(* PLC project Unnamed, Unknown Unnamed 1 *)
(* stored: creationDateTime 2025-06-21T03:07:53, modificationDateTime 2025-06-21T03:50:31 *)

PROGRAM ctud_pou
  VAR
    input1 AT %IX100.0 : BOOL;
    input2 AT %IX100.1 : BOOL;
    reset AT %IX100.2 : BOOL;
    load AT %IX100.3 : BOOL;
    output1 AT %QX100.0 : BOOL;
    output2 AT %QX100.1 : BOOL;
  END_VAR
  VAR
    CTUD0 : CTUD;
  END_VAR
  VAR  (* added by the conversion: wires and edge detectors of the diagram *)
    R_TRIG1 : R_TRIG;
    R_TRIG2 : R_TRIG;
  END_VAR

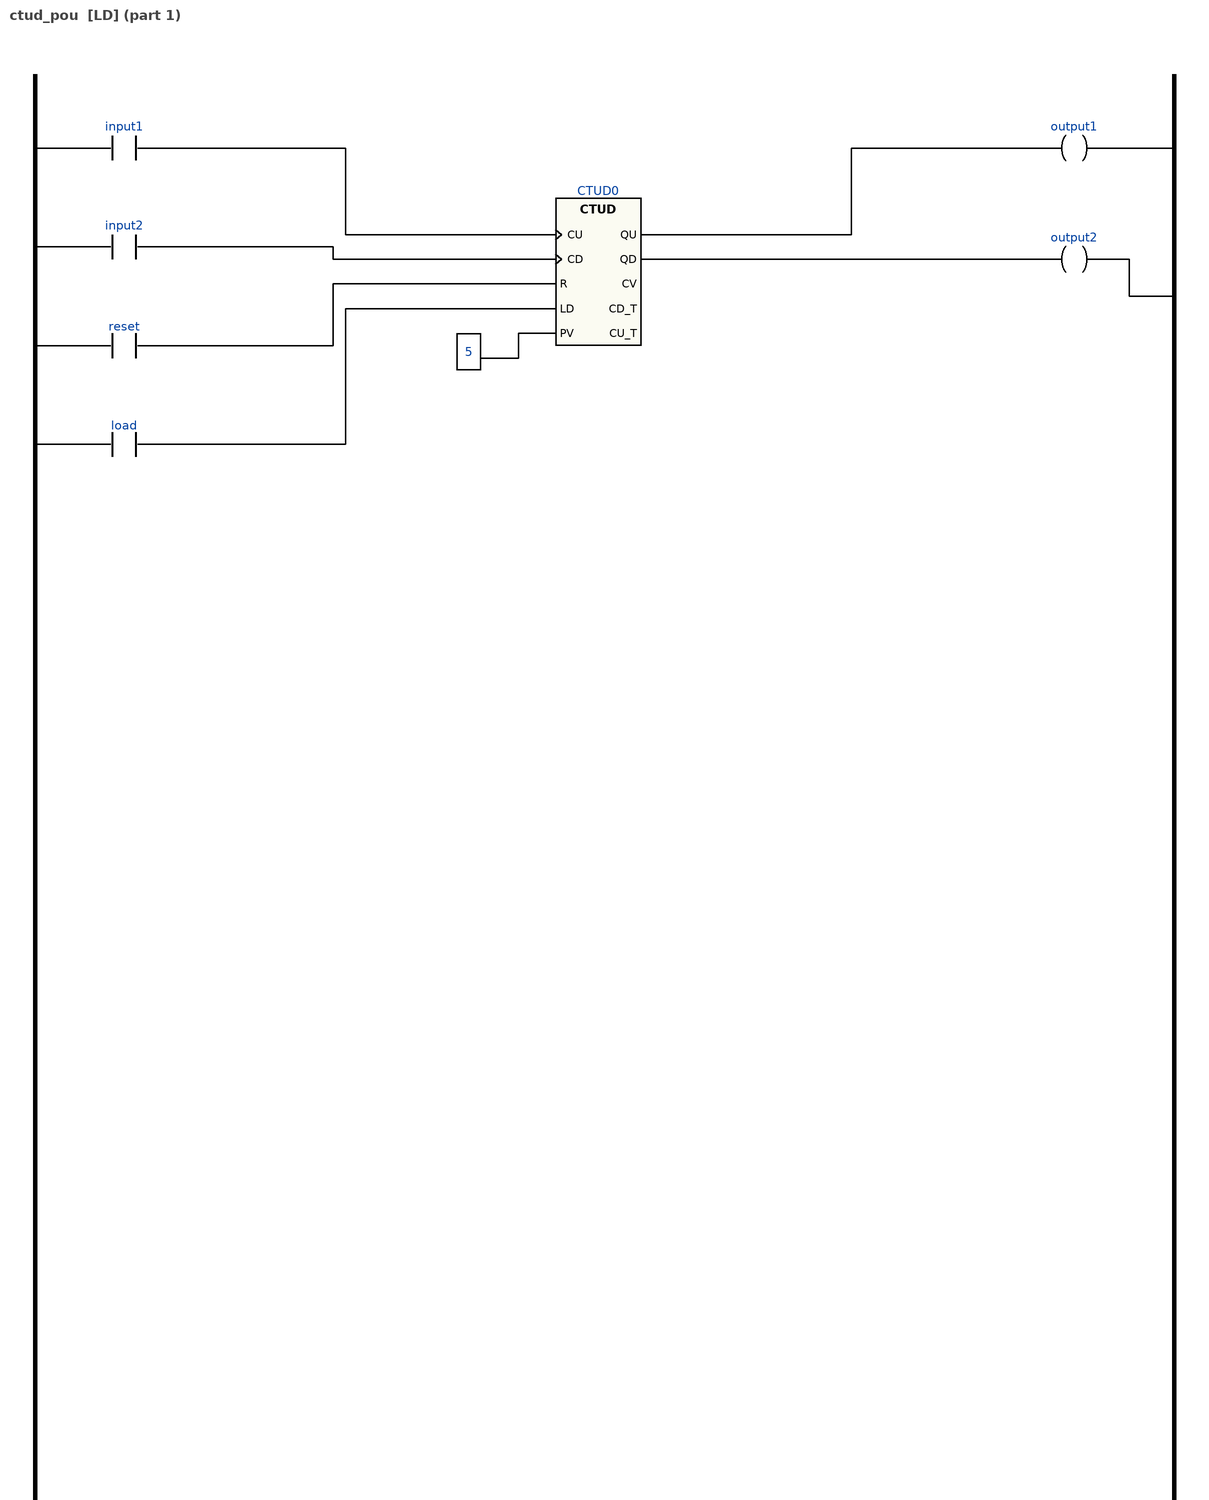
(* LD diagram, written out as Structured Text *)
R_TRIG1(CLK := input1);
R_TRIG2(CLK := input2);
CTUD0(CU := R_TRIG1.Q, CD := R_TRIG2.Q, R := reset, LD := load, PV := 5);
output1 := CTUD0.QU;
output2 := CTUD0.QD;
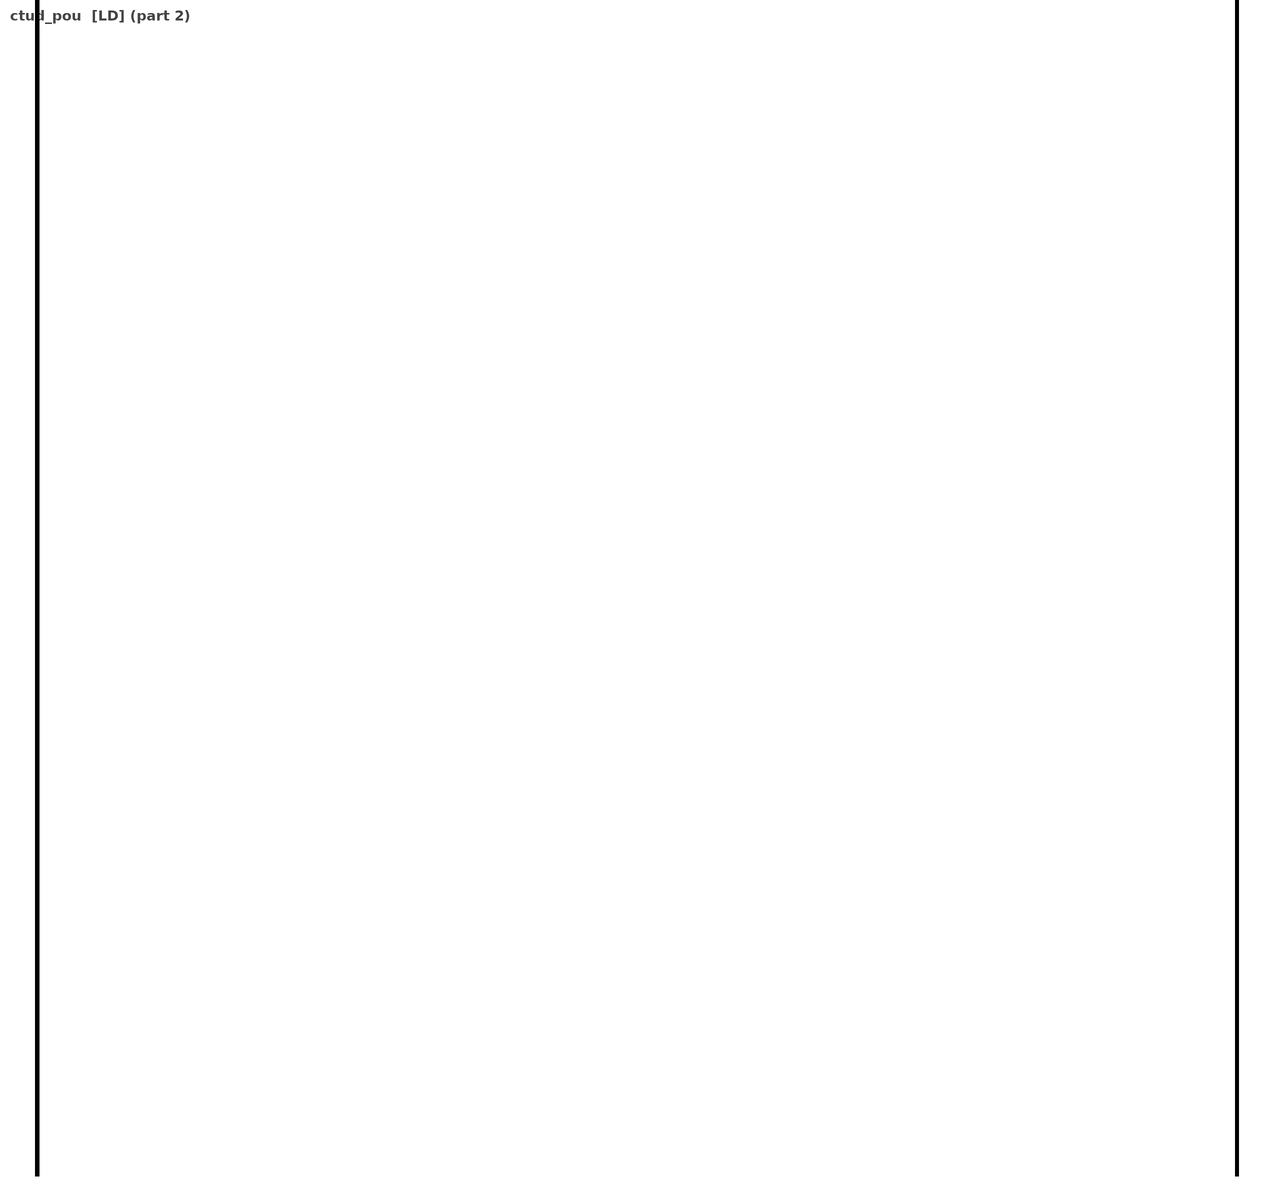
END_PROGRAM

CONFIGURATION Config0
  RESOURCE Res0 ON PLC
    TASK task0(INTERVAL := T#20ms, PRIORITY := 0);
    PROGRAM instance0 WITH task0 : ctud_pou;
  END_RESOURCE
END_CONFIGURATION
